INTERFACE I_Property

METHOD PUBLIC M_Add : BOOL
VAR_INPUT
	Name:			STRING(255);
	Value:			STRING(255);
END_VAR
END_METHOD

METHOD PUBLIC M_Reset
END_METHOD

END_INTERFACE

(* stored: Version 1.1.0.1
   Itf I_Property: Id {cbdabd9b-e5d6-0a5c-2592-22fbe23807be}
   Method M_Add: Id {536505c6-450b-0c0a-09ad-e54c0e4af995}
   Method M_Reset: Id {4633612c-6521-042e-27ef-3f71cf482de3} *)
